FUNCTION_BLOCK FB_Load_Following
VAR_INPUT
END_VAR
VAR_OUTPUT
END_VAR
VAR
	i: UINT;
	error_perc: REAL;
	delta: REAL; 
	reach_sp: FB_Reach_SP_ActP;
END_VAR

//  TO DO: valutare se, nel caso della potenza erogata dalla rete, conviene esprimere la potenza in termini percentuali rispetto alla potenza di rete
error_perc := ((GVL.VIRTUAL_POI_METER.active_power_prod - GVL_Load_Following.power_grid_max) / GVL_Load_Following.power_grid_max) * 100;

IF GVL.VIRTUAL_POI_METER.active_power_prod <= GVL_Load_Following.power_grid_min THEN
	
	delta := 0;
	GVL_Act_Pwr.total_sp := 0;

ELSIF (GVL.VIRTUAL_POI_METER.active_power_prod >= GVL_Load_Following.power_grid_min) AND (GVL.VIRTUAL_POI_METER.active_power_prod <= GVL_Load_Following.power_grid_max) THEN 
	
	delta := -1 *GVL_Load_Following.delta_fast;

ELSE

	delta := GVL_Load_Following.delta_fast;	

END_IF


IF (error_perc > 10) AND (error_perc < GVL_Load_Following.max_error_perc) THEN
	
	delta := GVL_Load_Following.delta_slow;

END_IF


IF error_perc < 10 THEN
	
	delta := 0;

END_IF

// TO DO: verificare se questa formula è corretta
GVL_Act_Pwr.total_sp := GVL_Act_Pwr.total_sp + delta * 0.100;   // + delta * dT con dT = tempo di esecuzione del main, pari a 100ms	
GVL_Act_Pwr.total_sp := MAX(0, MIN(1, GVL_Act_Pwr.total_sp)); 

reach_sp(sp_target_actp := GVL_Act_Pwr.total_sp);

END_FUNCTION_BLOCK

(* stored: Version 1.1.0.1, ProductVersion 3.1.4026.11
   POU FB_Load_Following: Id {99fe7c10-9c3c-44bf-b33b-9a1c48ebbc4b}, SpecialFunc None *)
